FUNCTION_BLOCK HAL


//--{attribute 'TcLinkTo' := 'TIID^Master (EtherCAT)^Term 1 (EK1200)^Term 7 (EL1008)^Channel 1^Input'}
//--     bVarIn2    AT%I*  : BOOL;  // linked via attribute

END_FUNCTION_BLOCK

(* stored: Version 1.1.0.1, ProductVersion 3.1.4024.12
   POU HAL: Id {3a9bd6e1-4674-4645-a5d3-1835b5ad1e40}, SpecialFunc None *)
